// TIA Portal V20 export
TYPE "typeDataFromSafety"
// stored: Access Published, IsFailsafeCompliant true, Namespace Safety
   STRUCT
      devicesSummary { ExternalWritable := 'False'} : "Safety.typeDevicesStatusSummary";   // General safety status of devices
      mainOp { ExternalWritable := 'False'} : "Safety.typeMainOpMode";   // Main Op State
      pHmi { ExternalWritable := 'False'} : "Safety.typePhmi";
      scsMode { ExternalWritable := 'False'} : "Safety.typeScsMode";   // SCS Mode
      rcMode1 { ExternalWritable := 'False'} : "Safety.typeRollChangeMode";   // Top Roll Change State
      rcMode2 { ExternalWritable := 'False'} : "Safety.typeRollChangeMode";   // Btm Roll Change State
      eStopStatus { ExternalWritable := 'False'} : "Safety.typeEstopStatus";   // E Stop Pressed
      fDoorSwitchStatus { ExternalWritable := 'False'} : "Safety.typeFDoorSwitchStatus";   // F Door Open Status
      fDoorCoilStatus { ExternalWritable := 'False'} : "Safety.typeFDoorUnlockOutput";   // F Door Unlock Cmd Status
      Zone1SafetyMainOpEnable { ExternalWritable := 'False'} : "Safety.typeSafetyOperationEnable";   // Zone1 Main Operation Enable
      Zone1SafetySubOpEnable { ExternalWritable := 'False'} : "Safety.typeSafetyOperationEnable";   // Zone1 Sub Operation Enable
      Zone2SafetyOpEnable { ExternalWritable := 'False'} : "Safety.typeSafetyOperationEnable";   // Zone2 Operation Enable
      Zone3SafetyOpEnable { ExternalWritable := 'False'} : "Safety.typeSafetyOperationEnable";   // Zone3 Operation Enable
      eStopZone1 { ExternalWritable := 'False'} : "Safety.typeEstopFunction";   // Safety status of estop button in Zone.1
      eStopZone2 { ExternalWritable := 'False'} : "Safety.typeEstopFunction";   // Safety status of estop button in Zone.2
      eStopZone3 { ExternalWritable := 'False'} : "Safety.typeEstopFunction";   // Safety status of estop button in Zone.3
      statusZone1 { ExternalWritable := 'False'} : "Safety.typeSafetyZoneStatus";   // Status of safety zone
      statusZone2 { ExternalWritable := 'False'} : "Safety.typeSafetyZoneStatus";   // Status of safety zone
      statusZone3 { ExternalWritable := 'False'} : "Safety.typeSafetyZoneStatus";   // Status of safety zone
      fDoorDrive { ExternalWritable := 'False'} : "Safety.typeFDoorFunction";
      driveStatus { ExternalWritable := 'False'} : "Safety.typeSafetyDriveStatus";
      SafetySensor { ExternalWritable := 'False'} : "Safety.typeSafetySensor";
      FeedbackFault { ExternalWritable := 'False'} : "Safety.typeFeedbackFault";
      AllEstopsOK { ExternalWritable := 'False'} : Bool;   // E Stop On Station All Ok
      allEstopButtonsOK { ExternalWritable := 'False'} : Bool;   // E Stop On Station All Ok
      AllEstopsOKfromOther { ExternalWritable := 'False'} : Bool;   // E Stop On Other Station All Ok
      AllFdoorClose { ExternalWritable := 'False'} : Bool;   // F Door All Closed
      AllSFDoorOpen { ExternalWritable := 'False'} : Bool;   // F Door Single Open
      AllMFDoorOpen { ExternalWritable := 'False'} : Bool;
      AnyNoMFDoorOpen { ExternalWritable := 'False'} : Bool;   // F Door No Multi Open
      safetyReleasedAllSafetyZones { ExternalWritable := 'False'} : Bool := false;   // All safety zones are released
      ackRequiredAnySafetyZone { ExternalWritable := 'False'} : Bool := false;   // At least one safety zone requires an acknowledge
      ackOP_changeRequired { ExternalWritable := 'False'} : Bool := false;   // ACK_OP is waiting for value change
      ackOperatorControlCondition : Bool;   // Ack Hmi Oprating Possible
      doorBoxAllReset : Bool;   // Combine All Door Box Reset Button
      totalSafetyReset { ExternalAccessible := 'False'; ExternalVisible := 'False'; ExternalWritable := 'False'} : Bool;   // Combine All Reset Trigger
      zone1DoorOpenRequest : Bool;   // Zone 1 Door Open Request
      zone2DoorOpenRequest : Bool;   // Zone 2 Door Open Request
      zone3DoorOpenRequest : Bool;   // Zone 3 Door Open Request
      zone1DriveAckReq : Bool;   // Zone 1 Safety Fault Ack Request
      zone2DriveAckReq : Bool;   // Zone 2 Safety Fault Ack Request
      zone3DriveAckReq : Bool;   // Zone 3 Safety Fault Ack Request
      noSafetyFault : Bool;   // All Zone No Safety Fault
      ConnectionBoxID { ExternalWritable := 'False'} : Int := 0;   // PHmi Connection Box ID
      BA60topTapeDoorForcedOpen : Bool;   // BA60 Top Tape Door Forced Open
      BA060STOP : Bool;   // Stop Done For BA060 Request
      BA60LightCurtainMuttingRequest : Bool;   // Light Curtain Mutting Request To BA060
      BA60LightCurtainDetect : Bool;   // BA060 Light Curtain Detect
      BA60RequestForEntry : Bool;   // Sepa Gripper Entry For Request From BA060
      BA60ExternalDoorOpen : Bool;
      BA60topTapeDoorNormalOpen : Bool;   // BA60 Top Tape Door Normal Open
      PhmiConnectedToBA60 : Bool;   // PHMI Connected Interface To BA60
      PhmiEnableToBA60 : Bool;   // PHMI Enable Interface To BA60
      HmiEnableToBA60 : Bool;   // Main OP HMI Enable Interface To BA60
      BA30CahodeCoverClose : Bool;
      BA30AnodeCoverClose : Bool;
      BA60Stacker1LightCurtainDetect : Bool;
      BA60Stacker1MaintenanceDoorOpen : Bool;
      SS1TimeExtension : Bool;
      EnableServoAck : Bool;
      SetupModFault : Bool;
      CathodeCoverSensorFault : Bool;
      AnodeCoverSensorFault : Bool;
      fDoor01UnlockPB : Bool;
      fDoor02UnlockPB : Bool;
      fDoor03UnlockPB : Bool;
      fDoor04UnlockPB : Bool;
      BA10 { ExternalWritable := 'False'} : "Safety.typeDataFlinkUsed";
      BA15 { ExternalWritable := 'False'} : "Safety.typeDataFlinkUsed";
      BA30 { ExternalWritable := 'False'} : "Safety.typeDataFlinkUsed";
      BA60 { ExternalWritable := 'False'} : "Safety.typeDataFlinkUsed";
      cvCoverStatus { ExternalWritable := 'False'} : "Safety.typeCvCoverStatus";
      hotWireCutterStatus { ExternalWritable := 'False'} : "Safety.typeHotWireCutter";
      fDoorUnwinderTopDoorOpenWarning { ExternalWritable := 'False'} : Bool;
      fDoorUnwinderBtmDoorOpenWarning { ExternalWritable := 'False'} : Bool;
      PhmiForcedDisconnection : Bool;
      CathodeConveyorCoverClosedCheck : Bool;
      AnodeConveyorCoverClosedCheck : Bool;
      FdoorForcedOpenStatus : "Safety.typeSafetyForcedDoorOpen";
   END_STRUCT;
END_TYPE
